PROGRAM NovramHandling
VAR
	fbReadSaveNovram:FB_NovRamReadWrite;
	stData:ST_NovramData;
END_VAR

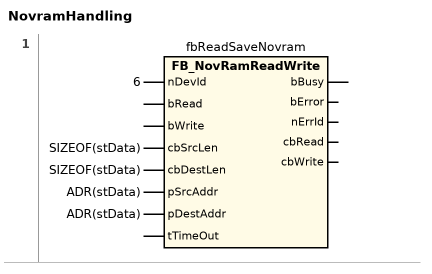
// NETWORK 1
fbReadSaveNovram(
    nDevId := 6,
    cbSrcLen := SIZEOF(stData),
    cbDestLen := SIZEOF(stData),
    pSrcAddr := ADR(stData),
    pDestAddr := ADR(stData)); // FB_NovRamReadWrite

END_PROGRAM

(* stored: Version 1.1.0.1, ProductVersion 3.1.4020.12
   POU NovramHandling: Id {caafbf8e-65ab-48bb-beec-4421fdf88665}, SpecialFunc None *)
